(* Logix 5000 project; controller IsaacExample 1769-L16ER-BB1B rev 32.11; software revision 32.00 *)

TASK MainTask (continuous, watchdog 500 ms) : MainProgram, Isaac_Interface

MODULES
   Local : 1769-L16ER-BB1B (PointIO 0, rev 32.11)
      Isaac_0 : vendor 1449 type 43 code 18 (Ethernet 192.168.2.93, rev 1.1, StandardDataDriven RPI 20 ms)
      Isaac_1 : vendor 1449 type 43 code 18 (Ethernet 192.168.2.94, rev 1.1, StandardDataDriven RPI 20 ms)
      Isaac_2 : vendor 1449 type 43 code 18 (Ethernet 192.168.2.95, rev 1.1, StandardDataDriven RPI 20 ms)
      Isaac_3 : vendor 1449 type 43 code 18 (Ethernet 192.168.2.96, rev 1.1, StandardDataDriven RPI 20 ms)
      Discrete_IO : Embedded (PointIO 1, rev 32.11, Output RPI 20 ms)
           Local:1:I.Data.1   // Red Push Btn
           Local:1:I.Data.2   // 2nd Green Btn
           Local:1:I.Data.0   // Green Btn
END_MODULES

TYPE Isaac_Tcp_Ip_Cfg :
STRUCT
   Status : DINT;   // Status
   Config_Capability : DINT;   // Capability
   Config_Control : DINT;   // IfCtrl
   Path_Size : INT;   // Epath
   Path : SINT[4];   // Padd
   IP_Address : DINT;   // IPAddr
   Network_Address : DINT;   // NetAddr
   Gateway_Address : DINT;   // GateWay
   Name_Server : DINT;   // DNS1
   Name_Server_2 : DINT;   // DNS2
   Domain_Name : STRING;   // Domain
   Host_Name : STRING;   // Host
   Safety_Network_Number : SINT[6];   // Ignore
   TTL : SINT;   // TTL
   Alloc_Control : SINT;   // MultCast
   Reserved : SINT;   // Reserved
   Num_Mcast : INT;   // MultCastAlloc
   Mcast_Start_Addr : DINT;   // MultCastStart
   Selected_Acd : BOOL;   // ACD
   Acd_Activity : SINT;   // ACDState
   Remote_MAC : SINT[6];   // MACRmt
   Arp_Pdu : SINT[28];   // ARP_PDU
   EthernetIP_Quick_Connect : BOOL;   // QuickCon
   Encp_Inactivity_Timeout : INT;   // InactTimeout
END_STRUCT
END_TYPE

TYPE IsaacCfg :
STRUCT
   AntiTie : SINT;   // AntiTie
   CurrentProgram : SINT;   // CurrentProgram
   ResultsOut : SINT;   // Results Out
   ResultsOutFraction : SINT;   // Results Out Fraction
   BaudRate : SINT;   // Baud Rate
   DataLogging : SINT;   // Data Logging
   PressureUnits : SINT;   // Pressure Units
   FlowUnits : SINT;   // Flow Units
   TestPresDigits : SINT;   // Test Pressure Digits
   ResultsPresDigits : SINT;   // Results Pressure Digits
   FlowPressureDigits : SINT;   // Flow Pressure Digits
   SpareCfg1 : SINT;   // SpareCfg1
   cosType : INT;   // ChangeOfState flags
   SpareCfg2 : SINT;   // SpareCfg2
   SpareCfg3 : SINT;   // SpareCfg3
END_STRUCT
END_TYPE

TYPE IsaacFirmwareCfg :
STRUCT
   CosType : INT;   // ChangeOfState Type
   ClassId : INT;   // ClassId
   Instance : INT;   // Instance
   Attribute : INT;   // Attribute
   LockPrgEdits : BOOL;   // LockPrgEdits
   LockCurrentPrgEdits : BOOL;   // LockCurrentPrgEdits
   LockCalibrationEdits : BOOL;   // LockCalibrationEdit
   ElectronicReg : BOOL;   // ElectronicReg
   ManualReg : BOOL;   // ManualReg
   Concurrent : BOOL;   // Concurrent
   BuzzerEnabled : BOOL;   // BuzzerEnabled
   BusyImm : BOOL;   // BusyImm
   DhcpEnabled : BOOL;   // DhcpEnabled
   OkToResetDevice : BOOL;   // OkToResetDevice
   LinkedFail : BOOL;   // LinkedFail
   HighBleed : BOOL;   // HighBleed
   ElectRegAlwaysOn : BOOL;   // ElectRegAlwaysOn
   SpareBit13 : BOOL;   // SpareBit_12
   SpareBit14 : BOOL;   // SpareBit_13
   SpareBit15 : BOOL;   // SpareBit_14
   TesterNumber : SINT;   // TesterNumber
   BaudRate : SINT;   // BaudRate
   DataLogging : SINT;   // DataLogging
   PressureUnits : SINT;   // PressUnts
   FlowUnits : SINT;   // FlowUnts
   TestPresDigits : SINT;   // TestDigits
   ResultsPresDigits : SINT;   // ResultsDigits
   FlowPresDigits : SINT;   // FlowDigits
   BCD : SINT;   // BCD
   NumberChannels : SINT;   // NumChans
   Sensors : SINT;   // Sensors
   AntiTie : SINT;   // LockedFlgs
   AvailTestTypes : SINT;   // AvailTestTypes
   SpareByte1 : SINT;   // SpareByte1
   SpareInt1 : INT;   // SpareInt1
   IoResetTime : INT;   // IoRstTime
   FilterPress : DINT;   // FilterPress
   FilterFlow : DINT;   // FilterFlow
   FilterFillSettle : DINT;   // FilterFillSettle
   FilterElectReg : DINT;   // FilterElectReg
   HighBleedPressure : INT;   // HighBleedPres
   SpareInt2 : INT;   // SpareInt2
   AtmPress : DINT;   // AtmPress
   SerialNumber : STRING_16;   // SerialNbr
   IpAddress : STRING_16;   // IpAddr
   IpNetmask : STRING_16;   // IpNetmask
   IpGateway : STRING_16;   // ipGateway
   MacAddress : STRING_20;   // MacAddr
   DateTime : STRING_20;   // DateTime
   ModelNumber : STRING_24;   // ModelNumber
   OptionsAndFittings : STRING_32;   // OptionsAndFittings
   SccsRevDate : STRING_24;   // SccsRevDate
   SccsRev : STRING_12;   // SccsRev
   SccsRevRange : STRING_24;   // SccsRevRange
END_STRUCT
END_TYPE

TYPE IsaacProgram :
STRUCT
   CosType : INT;   // ChangeOfState Type
   ClassId : INT;   // ClassId
   Instance : INT;   // Instance
   Attribute : INT;   // Attribute
   PrgNumb : SINT;   // PrgNumb
   SpareByte1 : SINT;   // SpareByte1
   Loops : INT;   // Loops
   PortEnabled1 : BOOL;   // PortEnabled1
   PortEnabled2 : BOOL;   // PortEnabled2
   PortEnabled3 : BOOL;   // PortEnabled3
   PortEnabled4 : BOOL;   // PortEnabled4
   FixtureValve1 : BOOL;   // FixtureValve1
   FixtureValve2 : BOOL;   // FixtureValve2
   ClampHoldFail : BOOL;   // ClampHoldFail
   Rslts232 : BOOL;   // Rslts232
   RsltsEthr : BOOL;   // RsltsEthr
   AutoFFill : BOOL;   // AutoFFill
   LeakStd : BOOL;   // LeakStd
   AutoVent : BOOL;   // AutoVent
   IncreaseLimit : BOOL;   // IncLimitEnbl
   EvalAtEnd : BOOL;   // EvalAtEnd
   ElectReg : BOOL;   // ElectReg
   SaveDacOnAbort : BOOL;   // SaveDaxOnAbort
   SpareBit_16 : BOOL;   // SpareBit_16
   SpareBit_17 : BOOL;   // SpareBit_17
   SpareBit_18 : BOOL;   // SpareBit_18
   SpareBit_19 : BOOL;   // SpareBit_19
   SpareBit_20 : BOOL;   // SpareBit_20
   SpareBit_21 : BOOL;   // SpareBit_21
   SpareBit_22 : BOOL;   // SpareBit_22
   SpareBit_23 : BOOL;   // SpareBit_23
   SpareBit_24 : BOOL;   // SpareBit_24
   SpareBit_25 : BOOL;   // SpareBit_25
   SpareBit_26 : BOOL;   // SpareBit_26
   SpareBit_27 : BOOL;   // SpareBit_27
   SpareBit_28 : BOOL;   // SpareBit_28
   SpareBit_29 : BOOL;   // SpareBit_29
   SpareBit_30 : BOOL;   // SpareBit_30
   SpareBit_31 : BOOL;   // SpareBit_31
   TestType : SINT;   // TestType
   NextPrg : SINT;   // NextPrg
   ElectRegDelay : SINT;   // ElectRegDelay
   SpareByte2 : SINT;   // SpareByte2
   TimeIdle : DINT;   // TimeIdle
   TimeClmp1 : DINT;   // TimeClmp1
   TimeClmp2 : DINT;   // TimeClmp2
   TimeFFill : DINT;   // TimeFFill
   TimeFill : DINT;   // TimeFill
   TimeSettle : DINT;   // TimeSettle
   TimeTest : DINT;   // TimeTest
   TimeVent : DINT;   // TimeVent
   TimeUnClmp1 : DINT;   // TimeUnClmp1
   TimeUnClmp2 : DINT;   // TimeUnClmp2
   SpareDInt1 : DINT;   // SpareDInt_1
   SpareDInt2 : DINT;   // SpareDInt_2
   TestPres : DINT;   // TestPres
   TestPresMin : DINT;   // RestPresMin
   TestPresMax : DINT;   // TestPresMax
   RegKp : DINT;   // RegKP
   RegKi : DINT;   // RegKi
   RegKd : DINT;   // RegKd
   PresFFill : DINT;   // PresFFill
   PresTestMin : DINT;   // PresTestMin
   PresTestMax : DINT;   // PresTestMax
   PresTestTrigger : DINT;   // PresTestTrigger
   Volume : DINT;   // Volume
   RampRate : DINT;   // RampRate
   SpareDInt3 : DINT;   // SpareDInt_3
   PrgName : STRING_16;   // PrgName
END_STRUCT
END_TYPE

TYPE STRING_12 :
STRUCT
   LEN : DINT;
   DATA : SINT[12];
END_STRUCT
END_TYPE

TYPE STRING_16 :
STRUCT
   LEN : DINT;
   DATA : SINT[16];
END_STRUCT
END_TYPE

TYPE STRING_20 :
STRUCT
   LEN : DINT;
   DATA : SINT[20];
END_STRUCT
END_TYPE

TYPE STRING_24 :
STRUCT
   LEN : DINT;
   DATA : SINT[24];
END_STRUCT
END_TYPE

TYPE STRING_32 :
STRUCT
   LEN : DINT;
   DATA : SINT[32];
END_STRUCT
END_TYPE

ADD_ON_INSTRUCTION EtherNetPathFix   (* revision 1.0, vendor Zaxis, Inc *)
VAR_IN_OUT
   Tester : IsaacTester; {required}
END_VAR
VAR_INPUT
   Start : DINT; {access Read Only, required}
END_VAR
VAR
   offsetToPath : INT; {access None}
   nullByte : STRING_12; {access Read Only}
   len : DINT; {access None}
END_VAR

ROUTINE Logic   (* ladder *)
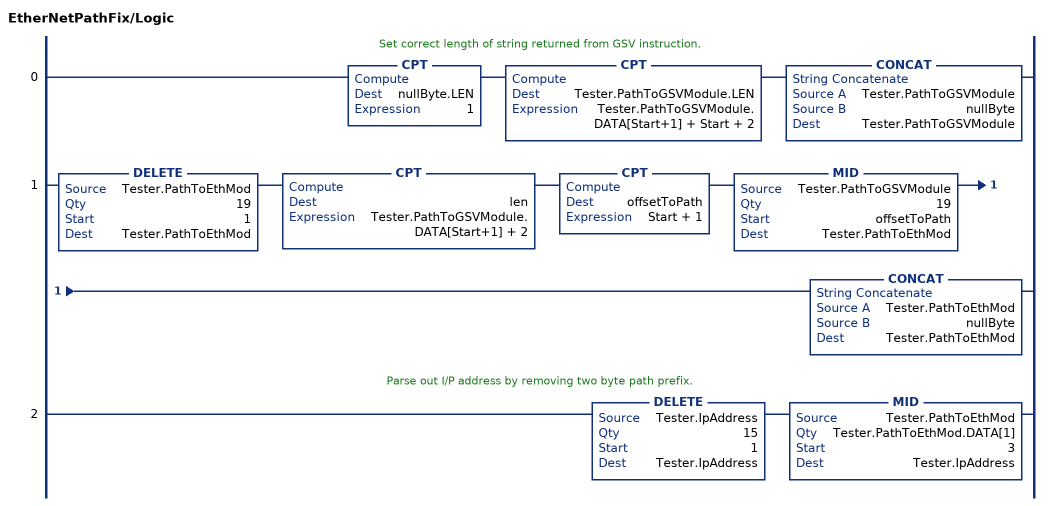
   // Set correct length of string returned from GSV instruction.
   0: CPT(nullByte.LEN,1)CPT(Tester.PathToGSVModule.LEN,Tester.PathToGSVModule.DATA[Start+1] + Start + 2)CONCAT(Tester.PathToGSVModule,nullByte,Tester.PathToGSVModule);
   1: DELETE(Tester.PathToEthMod,19,1,Tester.PathToEthMod)CPT(len,Tester.PathToGSVModule.DATA[Start+1] + 2)CPT(offsetToPath,Start + 1)MID(Tester.PathToGSVModule,19,offsetToPath,Tester.PathToEthMod)CONCAT(Tester.PathToEthMod,nullByte,Tester.PathToEthMod);
   // Parse out I/P address by removing two byte path prefix.
   2: DELETE(Tester.IpAddress,15,1,Tester.IpAddress)MID(Tester.PathToEthMod,Tester.PathToEthMod.DATA[1],3,Tester.IpAddress);
END_ROUTINE
END_ADD_ON_INSTRUCTION

ADD_ON_INSTRUCTION Isaac_Run   (* revision 1.0, vendor Zaxis, Inc *)
// Start Test
VAR_INPUT
   Start : BOOL; {access Read Only, required}   // Test Start
   AntiTie : BOOL; {access Read Only, required}   // AntiTie Bit
   AbortTest : BOOL; {access Read Only, required}   // Abort Bit
END_VAR
VAR_IN_OUT
   IT : IsaacTester; {required}
END_VAR
VAR_INPUT
   StartWInterlock : BOOL; {access Read Only, required}   // Start with Interlock
END_VAR

ROUTINE Logic   (* ladder *)
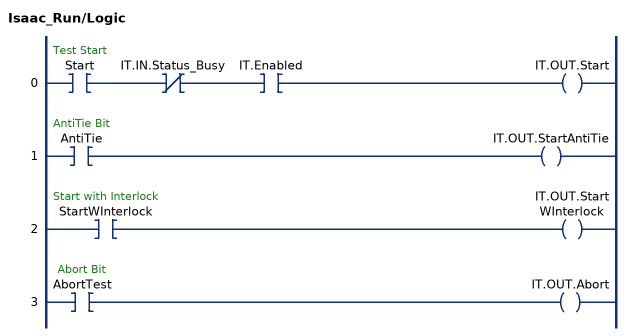
   0: XIC(Start)XIO(IT.IN.Status_Busy)XIC(IT.Enabled)OTE(IT.OUT.Start);
   1: XIC(AntiTie)OTE(IT.OUT.StartAntiTie);
   2: XIC(StartWInterlock)OTE(IT.OUT.StartWInterlock);
   3: XIC(AbortTest)OTE(IT.OUT.Abort);
END_ROUTINE
END_ADD_ON_INSTRUCTION

VAR_GLOBAL   (* controller tags *)
   Button_AntiTie : ALIAS FOR Local:1:I.Data.3;   // 2nd Red Button
   Button_Start : ALIAS FOR Local:1:I.Data.0;
   Button_StartWInterlock : ALIAS FOR Local:1:I.Data.2;
   Button_Stop : ALIAS FOR Local:1:I.Data.1;
   Isaac_Testers : IsaacTester[4] := ([0].Enabled := 1, [0].IpAddress := '$0D192.168.2.10', [0].PathToEthMod := '$00$12$0D192.168.2.10', [0].PathToGSVModule := '$10$00$12$0D192.168.2.100', [1].Enabled := 1, [2].Enabled := 1, [3].Enabled := 1);
   IsaacFirmware : IsaacFirmwareCfg;
   IsaacFirmware_Read : MESSAGE;
        MessageParameters(ServiceCode := 16#0001, DestinationTag := IsaacFirmware, ...)
   IsaacFirmware_Write : MESSAGE;
        .UnconnectedTimeout   // Timeout down to 3 seconds
        MessageParameters(ServiceCode := 16#0002, LocalElement := IsaacFirmware, ...)
   IsaacProgram : IsaacProgram;
   IsaacProgram_Read : MESSAGE;
        MessageParameters(ServiceCode := 16#0001, DestinationTag := IsaacProgram, ...)
   IsaacProgram_Write : MESSAGE;
        MessageParameters(ServiceCode := 16#0002, LocalElement := IsaacProgram, ...)
   IsaacTcp_Ip_Read : MESSAGE;
        MessageParameters(ServiceCode := 16#0001, DestinationTag := IsaacTcpIp_Cfg, ...)
   IsaacTcp_Ip_Write : MESSAGE;
        MessageParameters(ServiceCode := 16#0002, LocalElement := IsaacTcpIp_Cfg, ...)
   IsaacTcpIp_Cfg : Isaac_Tcp_Ip_Cfg;
   TCP_IP_Write : BOOL;
END_VAR

PROGRAM Isaac_Interface   (* main routine Isaac_Run *)
VAR
   Debug : BOOL;
   Debug2 : BOOL;
   EtherNetPathGet : EtherNetPathFix := (Start := 2);
   Firmware_Read : BOOL;
   Firmware_Write : BOOL;
   FirmwareSetup_DN : BOOL;
   FirmwareSetup_EN : BOOL;   // Firmware Setup Started
   Idx : DINT;
   InitialSetup_Do : BOOL;
   Isaac_Configuration : IsaacCfg := (CurrentProgram := 1, BaudRate := 4, DataLogging := 1, PressureUnits := 1, TestPresDigits := 3, ResultsPresDigits := 5, FlowPressureDigits := 3); {access None}
   Isaac_FirmwareSetup_DN : BOOL;
   Isaac_InitializeProgram : BOOL := 1;
   IT_Idx : DINT := 1;
   IT_Size : DINT := 3;
   Program_Read : BOOL;
   Program_Write : BOOL;
   Run_Enabled : BOOL := 1;
   Setup_Step_1 : BOOL;
   Setup_Step_2 : BOOL;
   Setup_Step_3 : BOOL;
   StartTest : Isaac_Run;
   TCP_IP_Read : BOOL;
   Temp : BOOL := 1;
   Tester : IsaacTester := (Enabled := 1);
END_VAR
VAR_INPUT
   Name : STRING; {access Read Only}
END_VAR

ROUTINE Isaac_FirmwareSetup   (* ladder *)
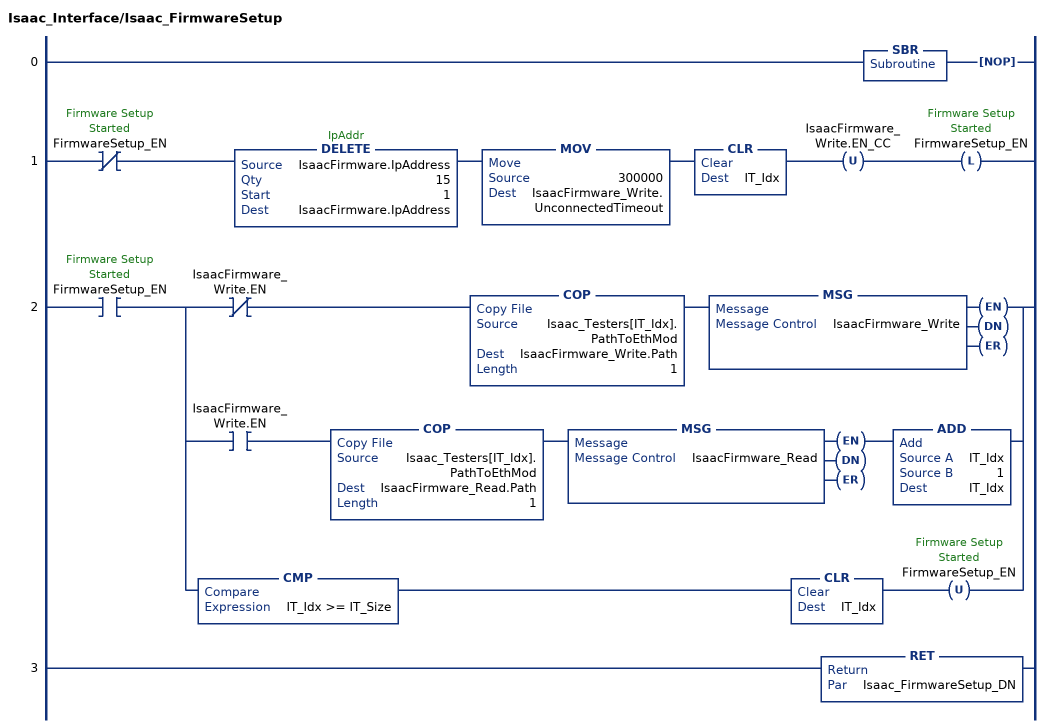
   0: SBR()NOP();
   1: XIO(FirmwareSetup_EN)DELETE(IsaacFirmware.IpAddress,15,1,IsaacFirmware.IpAddress)MOV(300000,IsaacFirmware_Write.UnconnectedTimeout)CLR(IT_Idx)OTU(IsaacFirmware_Write.EN_CC)OTL(FirmwareSetup_EN);
   2: XIC(FirmwareSetup_EN)[XIO(IsaacFirmware_Write.EN) COP(Isaac_Testers[IT_Idx].PathToEthMod,IsaacFirmware_Write.Path,1) MSG(IsaacFirmware_Write) ,XIC(IsaacFirmware_Write.EN) COP(Isaac_Testers[IT_Idx].PathToEthMod,IsaacFirmware_Read.Path,1) MSG(IsaacFirmware_Read) ADD(IT_Idx,1,IT_Idx) ,CMP(IT_Idx >= IT_Size) CLR(IT_Idx) OTU(FirmwareSetup_EN) ];
   3: RET(Isaac_FirmwareSetup_DN);
END_ROUTINE

ROUTINE Isaac_Initialize   (* ladder *)
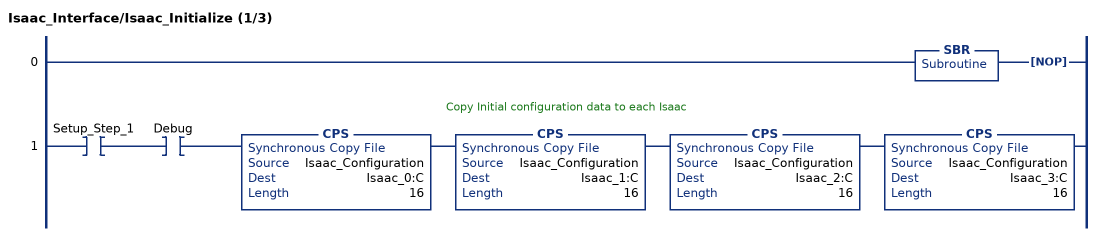
   0: SBR()NOP();
   // Copy Initial configuration data to each Isaac
   1: XIC(Setup_Step_1)XIC(Debug)CPS(Isaac_Configuration,Isaac_0:C,16)CPS(Isaac_Configuration,Isaac_1:C,16)CPS(Isaac_Configuration,Isaac_2:C,16)CPS(Isaac_Configuration,Isaac_3:C,16);
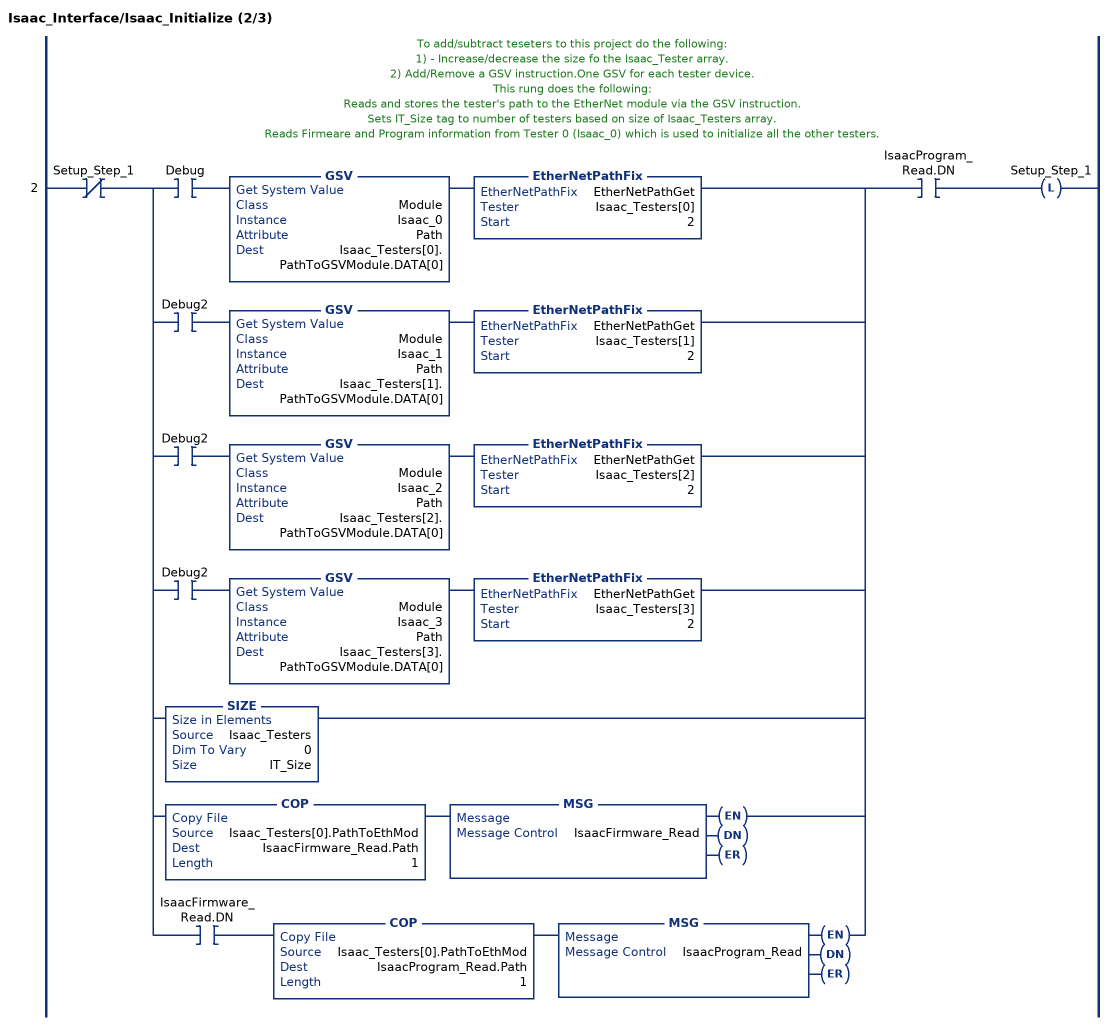
   // To add/subtract teseters to this project do the following:
   // 1) - Increase/decrease the size fo the Isaac_Tester array.
   // 2) Add/Remove a GSV instruction.One GSV for each tester device.
   // This rung does the following:
   // Reads and stores the tester's path to the EtherNet module via the GSV instruction.
   // Sets IT_Size tag to number of testers based on size of Isaac_Testers array.
   // Reads Firmeare and Program information from Tester 0 (Isaac_0) which is used to initialize all the other testers.
   2: XIO(Setup_Step_1)[XIC(Debug) GSV(Module,Isaac_0,Path,Isaac_Testers[0].PathToGSVModule.DATA[0]) EtherNetPathFix(EtherNetPathGet,Isaac_Testers[0],2) ,XIC(Debug2) GSV(Module,Isaac_1,Path,Isaac_Testers[1].PathToGSVModule.DATA[0]) EtherNetPathFix(EtherNetPathGet,Isaac_Testers[1],2) ,XIC(Debug2) GSV(Module,Isaac_2,Path,Isaac_Testers[2].PathToGSVModule.DATA[0]) EtherNetPathFix(EtherNetPathGet,Isaac_Testers[2],2) ,XIC(Debug2) GSV(Module,Isaac_3,Path,Isaac_Testers[3].PathToGSVModule.DATA[0]) EtherNetPathFix(EtherNetPathGet,Isaac_Testers[3],2) ,SIZE(Isaac_Testers,0,IT_Size) ,COP(Isaac_Testers[0].PathToEthMod,IsaacFirmware_Read.Path,1) MSG(IsaacFirmware_Read) ,XIC(IsaacFirmware_Read.DN) COP(Isaac_Testers[0].PathToEthMod,IsaacProgram_Read.Path,1) MSG(IsaacProgram_Read) ]XIC(IsaacProgram_Read.DN)OTL(Setup_Step_1);
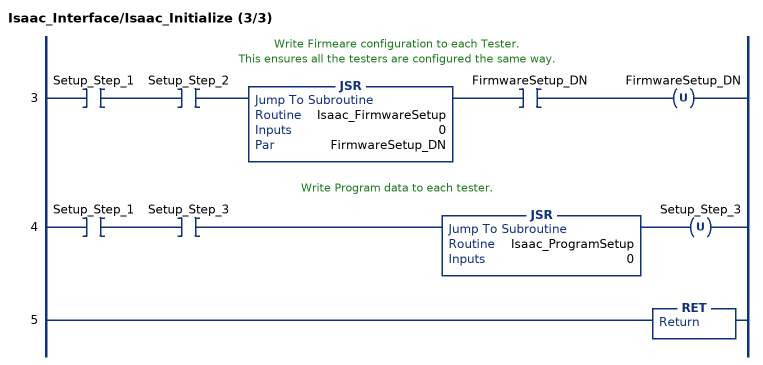
   // Write Firmeare configuration to each Tester.
   // This ensures all the testers are configured the same way.
   3: XIC(Setup_Step_1)XIC(Setup_Step_2)JSR(Isaac_FirmwareSetup,0,FirmwareSetup_DN)XIC(FirmwareSetup_DN)OTU(FirmwareSetup_DN);
   // Write Program data to each tester.
   4: XIC(Setup_Step_1)XIC(Setup_Step_3)JSR(Isaac_ProgramSetup,0)OTU(Setup_Step_3);
   5: RET();
END_ROUTINE

ROUTINE Isaac_MapInputs   (* ladder *)
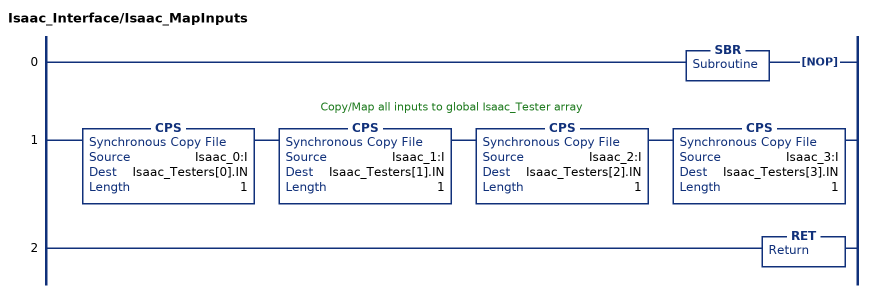
   0: SBR()NOP();
   // Copy/Map all inputs to global Isaac_Tester array
   1: CPS(Isaac_0:I,Isaac_Testers[0].IN,1)CPS(Isaac_1:I,Isaac_Testers[1].IN,1)CPS(Isaac_2:I,Isaac_Testers[2].IN,1)CPS(Isaac_3:I,Isaac_Testers[3].IN,1);
   2: RET();
END_ROUTINE

ROUTINE Isaac_MapOutputs   (* ladder *)
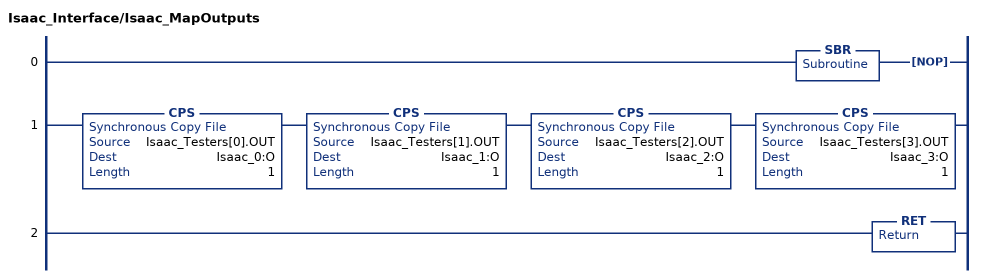
   0: SBR()NOP();
   1: CPS(Isaac_Testers[0].OUT,Isaac_0:O,1)CPS(Isaac_Testers[1].OUT,Isaac_1:O,1)CPS(Isaac_Testers[2].OUT,Isaac_2:O,1)CPS(Isaac_Testers[3].OUT,Isaac_3:O,1);
   2: RET();
END_ROUTINE

ROUTINE Isaac_ProgramSetup   (* ladder *)
   0: NOP();
END_ROUTINE

ROUTINE Isaac_Run   (* ladder *)
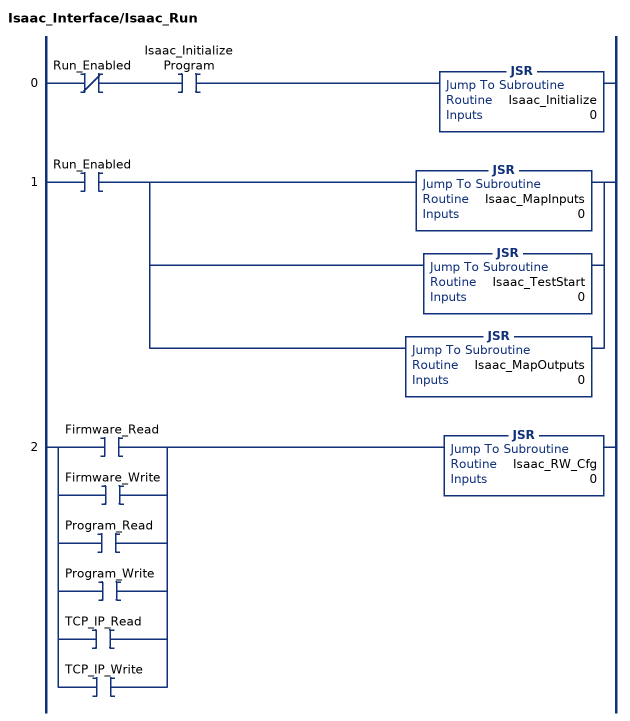
   0: XIO(Run_Enabled)XIC(Isaac_InitializeProgram)JSR(Isaac_Initialize,0);
   1: XIC(Run_Enabled)[JSR(Isaac_MapInputs,0) ,JSR(Isaac_TestStart,0) ,JSR(Isaac_MapOutputs,0) ];
   2: [XIC(Firmware_Read) ,XIC(Firmware_Write) ,XIC(Program_Read) ,XIC(Program_Write) ,XIC(TCP_IP_Read) ,XIC(TCP_IP_Write) ]JSR(Isaac_RW_Cfg,0);
END_ROUTINE

ROUTINE Isaac_RW_Cfg   (* ladder *)
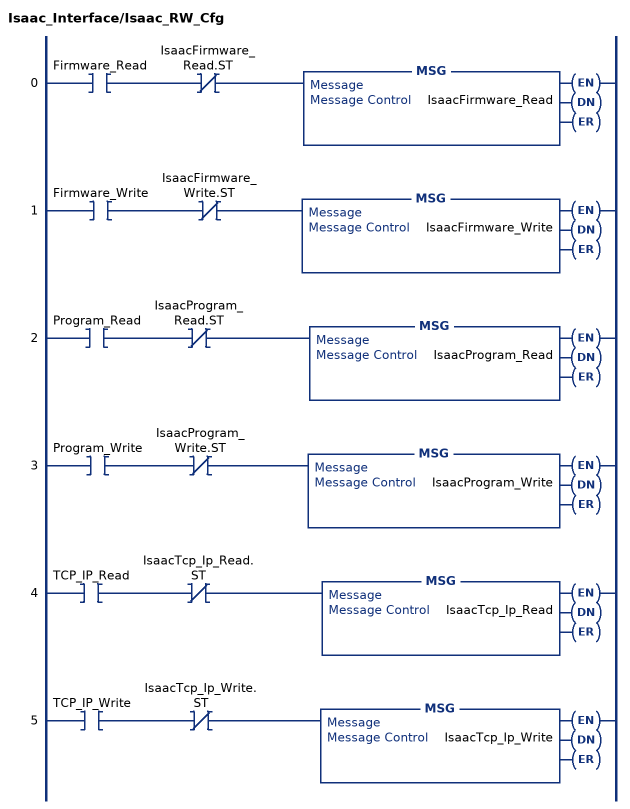
   0: XIC(Firmware_Read)XIO(IsaacFirmware_Read.ST)MSG(IsaacFirmware_Read);
   1: XIC(Firmware_Write)XIO(IsaacFirmware_Write.ST)MSG(IsaacFirmware_Write);
   2: XIC(Program_Read)XIO(IsaacProgram_Read.ST)MSG(IsaacProgram_Read);
   3: XIC(Program_Write)XIO(IsaacProgram_Write.ST)MSG(IsaacProgram_Write);
   4: XIC(TCP_IP_Read)XIO(IsaacTcp_Ip_Read.ST)MSG(IsaacTcp_Ip_Read);
   5: XIC(TCP_IP_Write)XIO(IsaacTcp_Ip_Write.ST)MSG(IsaacTcp_Ip_Write);
END_ROUTINE

ROUTINE Isaac_TestStart   (* ladder *)
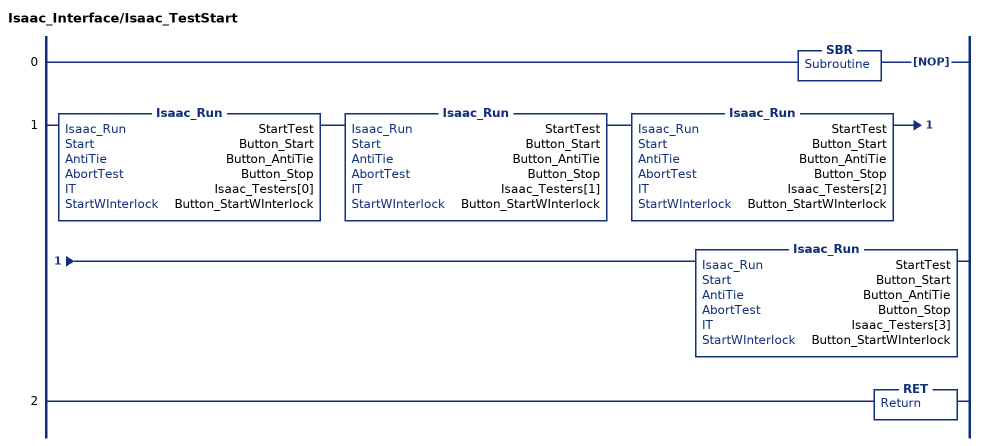
   0: SBR()NOP();
   1: Isaac_Run(StartTest,Button_Start,Button_AntiTie,Button_Stop,Isaac_Testers[0],Button_StartWInterlock)Isaac_Run(StartTest,Button_Start,Button_AntiTie,Button_Stop,Isaac_Testers[1],Button_StartWInterlock)Isaac_Run(StartTest,Button_Start,Button_AntiTie,Button_Stop,Isaac_Testers[2],Button_StartWInterlock)Isaac_Run(StartTest,Button_Start,Button_AntiTie,Button_Stop,Isaac_Testers[3],Button_StartWInterlock);
   2: RET();
END_ROUTINE
END_PROGRAM

PROGRAM MainProgram   (* main routine MainRoutine *)

ROUTINE MainRoutine   (* ladder *)
END_ROUTINE
END_PROGRAM
